# EPICS autosave request: iocs/QHYIOC/iocBoot/iocQHY/auto_settings.req
file "QHY_settings.req",       P=$(P),  R=cam1:
file "NDStdArrays_settings.req",  P=$(P),  R=image1:
file "commonPlugin_settings.req", P=$(P)
